Staubli VAL3: remSetStagePos.pgx

program remSetStagePos(string& sArgs[] (dimensions=1), string& sReturn[] (dimensions=1))
begin
  // Set the PPS status in the robot
  //
  logMsg("call remSetStagePos")
  call remSetnGlobal(sArgs,nStagePos,-50000,50000,"NOTSTAGEPOS",sReturn)
end
